// TIA Portal project "Motor_Fault_Detection_Alarm_System" (V18)

(* hardware
DEVICE "S7-1200 station_1"  S7-1200 Station
   slot 0: "Rack_0"  S7-1200 Rack  Rack  V1.0
   slot 1: "PLC_1"  CPU 1214C DC/DC/DC  6ES7 214-1AG40-0XB0  V4.6
*)

// ===== PLC "PLC_1"  CPU 1214C DC/DC/DC =====

VAR_GLOBAL   // PLC tag table "Default tag table"
   "Start_PB" AT %I0.0 : Bool;
   "Stop_PB" AT %I0.1 : Bool;
   "Temp_Fault" AT %I0.2 : Bool;
   "Ack_PB" AT %I0.3 : Bool;
   "Reset_PB" AT %I0.4 : Bool;
   "Motor_Run" AT %Q0.0 : Bool;
   "Alarm_Light" AT %Q0.1 : Bool;
   "Buzzer" AT %Q0.2 : Bool;
   "Motor_Latch" AT %M0.0 : Bool;
   "Fault_Latch" AT %M0.1 : Bool;
   "Alarm_Ack" AT %M0.2 : Bool;
END_VAR

ORGANIZATION_BLOCK "Main"   // OB1, LAD, ProgramCycle
TITLE = "Main Program Sweep (Cycle)"
{ S7_Optimized_Access := 'TRUE' }
VERSION : 0.1
   VAR_INPUT
      Initial_Call : Bool;   // Initial call of this OB
      Remanence : Bool;   // =True, if remanent data are available
   END_VAR
BEGIN

REGION Network 1: Motor Latch
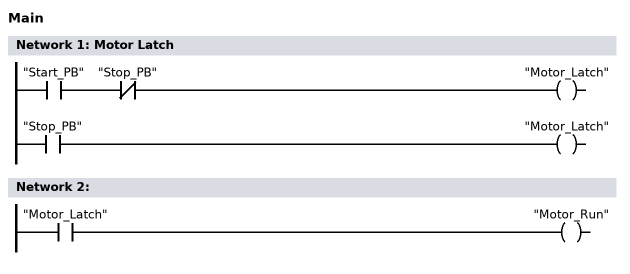
   RUNG wire#powerrail
      Contact( "Start_PB" )
      I_Contact( "Stop_PB" )
      Coil( "Motor_Latch" )
   END_RUNG
   RUNG wire#powerrail
      Contact( "Stop_PB" )
      Coil( "Motor_Latch" )
   END_RUNG
   // the same network as SCL:
   "Motor_Latch" := "Start_PB" AND NOT "Stop_PB";
   "Motor_Latch" := "Stop_PB";
END_REGION

REGION Network 2
   RUNG wire#powerrail
      Contact( "Motor_Latch" )
      Coil( "Motor_Run" )
   END_RUNG
   // the same network as SCL:
   "Motor_Run" := "Motor_Latch";
END_REGION
END_ORGANIZATION_BLOCK